INTERFACE IRegulator

METHOD M_Active : UINT
VAR_INPUT
	(* controller input  *)
	fSetpointValue			: LREAL;		// setpoint value
	fActualValue			: LREAL;		// actual value
	bReset					: BOOL;			// reset flag
	(* controller values *)
	stRegParams				: ST_RegParams;
END_VAR
VAR_OUTPUT
	fCtrlOutput				: LREAL;		// controller output command
END_VAR
END_METHOD

PROPERTY P_Error : BOOL
GET
END_GET
SET
END_SET
END_PROPERTY

END_INTERFACE

(* stored: Version 1.1.0.1, ProductVersion 3.1.4024.11
   Itf IRegulator: Id {32a4efb6-a6ad-4b6b-a70b-dce0caacc678}
   Method M_Active: Id {6a44f168-9b77-4c09-94c4-f2895005834c}
   Property P_Error: Id {cfd9924e-7f8a-4801-b7c3-48c3289e5279}
   Get Get: Id {b64430ec-3f38-4f9f-a2e7-985cd8915753}
   Set Set: Id {b8d23d20-be54-4d31-8fc3-250f7e1dbd65} *)
